PROGRAM MAIN
VAR
	
	a1			:INT		:=100;
	b2			:BOOL		:=FALSE;
	c3 			:LREAL 		:= 0;
	
	er			:DWORD;
	er1         :DWORD;
	
	arrLeftBoxStack	:ARRAY[1..50] OF BOX;
	arrRightBoxStack:ARRAY[1..50] OF BOX;
	
	
	//er:=axis_SmallGate_Left.NcToPlc.StateDWord

END_VAR

axis_BigGate_Left();	
er := axis_BigGate_Left.NcToPlc.StateDWord AND SHL(16#1, 28);
er1:= axis_BigGate_Left.NcToPlc.StateDWord AND SHL(16#1, 31);

END_PROGRAM

(* stored: Version 1.1.0.1, ProductVersion 3.1.4024.14
   POU MAIN: Id {4c1d16d0-3590-4597-9505-643a192836e5}, SpecialFunc None *)
